Staubli VAL3: onEnterEvent.pgx

program onEnterEvent()
  local string l_sPath
begin
  //
  if saveData:mode>0 and sEvent!=""
    call loadPage("instruction/PROG/page_instr",sEvent)
  endIf
  //
end
